FUNCTION F_map : REAL
VAR_INPUT
	// input variables
	fValue : REAL; // 16000
	fInMin : REAL; // 0
	fInMax : REAL; // 32767
	fOutMin: REAL; // 100
	fOutMax: REAL; // 0
END_VAR
VAR
	// internal variables
END_VAR

// map fValue linearly from [fInMin, fInMAx] to [fOutMin, fOutMax]

F_map := fOutMin + (fValue - fInMin)*(fOutMax-fOutMin)/(fInMax-fInMin);

END_FUNCTION

(* stored: Version 1.1.0.1, ProductVersion 3.1.4024.6
   POU F_map: Id {a5d038bb-31a5-4c9a-a99a-31e10298b8be}, SpecialFunc None *)
